FUNCTION F_DumpChiller_Error : FB_DumpChiller
VAR_INPUT
END_VAR
VAR
	fbDumpChiller : FB_DumpChiller;
END_VAR

fbDumpChiller(
	bAmphosOn := TRUE,
	bDumpChillerFlow := FALSE
);
F_DumpChiller_Error := fbDumpChiller;

END_FUNCTION

(* stored: Version 1.1.0.1, ProductVersion 3.1.4020.14
   POU F_DumpChiller_Error: Id {58e23adf-f2cb-4323-9c7d-f5f434c77017}, SpecialFunc None *)
